PROGRAM MAIN
VAR
	NonPersMainVarBool1:BOOL:=TRUE;
	NonPersMainVarBool2:BOOL:=FALSE;
	TestFB1_DB1:TestFB1;
	
	fbToLocal 		: FB_FileTimeToTzSpecificLocalTime;
	fileTime        : T_FILETIME;
	fbGetSystemTime : GETSYSTEMTIME;
END_VAR
VAR PERSISTENT
	PersMainVarBool3:BOOL:=TRUE;
	PersMainVarBool4:BOOL:=FALSE;
	PersMainVarInt1:INT:=0;
END_VAR


PersMainVarInt1:=PersMainVarInt1+1;
TestFB1_DB1(I_Run:=TRUE);

fbGetSystemTime(timeLoDW=>fileTime.dwLowDateTime, timeHiDW=>fileTime.dwHighDateTime );
GVL.DatetimeUTC := FILETIME_TO_DT(fileTime);
fbToLocal( in := fileTime, tzInfo := WEST_EUROPE_TZI );
GVL.Datetime := FILETIME_TO_DT( fbToLocal.out );
GVL.ActualDate := DT_TO_DATE(GVL.Datetime);
GVL.ActualTime := DT_TO_TIME(GVL.Datetime);
GVL.ActualLTime := TIME_TO_LTIME(GVL.ActualTime);

END_PROGRAM

(* stored: Version 1.1.0.1, ProductVersion 3.1.4024.4
   POU MAIN: Id {257901d8-cca3-4506-9fdf-a810e9ab7fed}, SpecialFunc None *)
